ABB RobotStudio station: GJJRobotStudioAss1005f.rspag

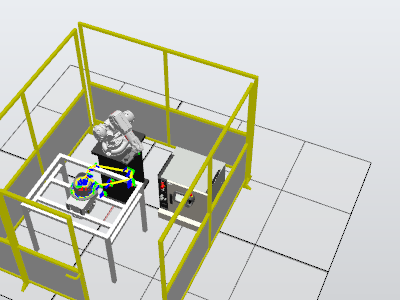
--- station ---
Station GJJAssessment1 (saved by RobotStudio 23.3.10550.0)
Controller Controller1
  mechanical unit ROB_1: IRB140_6_81_C_03, 6 joints, base frame (0, 0, 1000) mm
  mechanical unit M7DM1: MTD_250_M2009_REV1_01, 1 joints, base frame (769.44, 0, 1044.6) mm, rotated rx 0 ry 0 rz 180 deg
Layout (positions relative to the parent item):
  - IRB140_6_81_C_03 [mechanism, from %ABB.RobotStudio.Models.IRB140%\IRB140_6_81_C_G_03.rslib] at (0, 0, 1000) mm; joint values [-1.8898, -0.7873, -3.0781, -1.6729, -1.4587, 5.439] (rad or m)
  - MTD_250_M2009_REV1_01 [mechanism, from %ABB.RobotStudio.Models.GearUnits%\MTD_250_M2009_REV1_01.rslib] at (769.44, 0, 1044.6) mm, rotated rx 0 ry 0 rz 180 deg; joint values [19.7219] (rad or m)
  - potty1 [part] at (720.18, 192.49, 1031.85) mm, rotated rx 90 ry 0 rz 49.98 deg, size 275.1 x 194.8 x 257.3 mm
  - holder [part] at (392.98, 450, 1000) mm, rotated rx 90 ry 0 rz 0 deg, size 50 x 120 x 49.5 mm
  - SmartComponent_1_3 [smart component, from Libraries\SmartComponent_1.rslib] at (211.42, 435.22, 1354.55) mm, rotated rx -59.69 ry 89.8 rz -69.29 deg
      connections:
        SmartComponent_1_3.Closegrippers -> Attacher.Execute
        SmartComponent_1_3.Opengrippers -> Detacher.Execute
    - MyNewToolwithoutpen [mechanism, from Libraries\SmartComponent_1.rslib] at (0, 0, 0) mm
    - Attacher [smart component, from Components\Attacher.rslib]
        properties: Parent=MyNewToolwithoutpen; Flange=0; Child=The_Pen; Mount=false; Offset=[0 0 0]; Orientation=[0 0 0]
    - Detacher [smart component, from Components\Detacher.rslib]
        properties: Child=The_Pen; KeepPosition=false
  - The_Pen [part] at (215.35, 450.26, 1184.42) mm, rotated rx -90 ry 0 rz -90 deg, size 50 x 143 x 50 mm
  - Fence_2500 [graphiccomponentgroup, from Equipment\Fence_2500.rslib] at (1625.03, -938.91, 0) mm, rotated rx 0 ry 0 rz 90 deg
    - Body 1 [part, from Equipment\Fence_2500.rslib]
    - Body 2 [part, from Equipment\Fence_2500.rslib]
  - Fence_2500_2 [graphiccomponentgroup, from Equipment\Fence_2500.rslib] at (1620.42, 1504.32, 0) mm, rotated rx 0 ry 0 rz 90 deg
    - Body 1 [part, from Equipment\Fence_2500.rslib]
    - Body 2 [part, from Equipment\Fence_2500.rslib]
  - Fence_2500_3 [graphiccomponentgroup, from Equipment\Fence_2500.rslib] at (-975.12, -948, 0) mm
    - Body 1 [part, from Equipment\Fence_2500.rslib]
    - Body 2 [part, from Equipment\Fence_2500.rslib]
  - Gate [graphiccomponentgroup, from Equipment\Fence_Gate.rslib] at (1749.55, -943.09, 0) mm
    - Body 1 [part, from Equipment\Fence_Gate.rslib]
    - Body 2 [part, from Equipment\Fence_Gate.rslib]
    - Body 3 [part, from Equipment\Fence_Gate.rslib]
  - FlexPendant [part, from %ABB.RobotStudio.Models.IRC5%\FlexPendant.rslib] at (227.42, 1060.08, 778.08) mm, rotated rx -20.58 ry 0 rz 90 deg
  - MTDTable_Group [graphiccomponentgroup] at (367.09, -596.22, 0) mm
    - Height1 [part] at (850, 0, 0) mm, size 50 x 50 x 1000 mm
    - Height1_2 [part] at (850, 1150, 0) mm, size 50 x 50 x 1000 mm
    - Height1_3 [part] at (0, 1150, 0) mm, size 50 x 50 x 1000 mm
    - Height1_4 [part], size 50 x 50 x 1000 mm
    - Length1 [part] at (603.96, 0, 790) mm, size 50 x 1200 x 50 mm
    - Length1_2 [part] at (284.07, 0, 790) mm, size 50 x 1200 x 50 mm
    - Length1_3 [part] at (850, 0, 950) mm, size 50 x 1200 x 50 mm
    - Length1_4 [part] at (0, 0, 950) mm, size 50 x 1200 x 50 mm
    - Width1 [part] at (0, 0, 950) mm, size 900 x 50 x 50 mm
    - Width1_2 [part] at (0, 1150, 950) mm, size 900 x 50 x 50 mm
    - Width1_3 [part] at (0, 1150, 790) mm, size 900 x 50 x 50 mm
    - Width1_4 [part] at (0, 0, 790) mm, size 900 x 50 x 50 mm
  - IRC5_Singel-Cabinet [part, from %ABB.RobotStudio.Models.IRC5%\IRC5_Singel-Cabinet.rslib] at (-8.18, 1022.3, 100) mm, rotated rx 90 ry 0 rz 90 deg
  - RobotTable_Group [graphiccomponentgroup] at (-370.74, -2173.9, 0) mm
    - Bottom [part] at (0, 1929.69, 0) mm, size 550 x 500 x 50 mm
    - Top [part] at (0, 1929.69, 950) mm, size 550 x 500 x 50 mm
    - Table [part] at (46.03, 1981.79, 0) mm, size 450 x 400 x 1000 mm
Attachment: potty1 is attached to MTD_250_M2009_REV1_01 / Link1
Attachment: SmartComponent_1_3 is attached to IRB140_6_81_C_03 / Link6
Station logic (signal -> signal, property => property):
  Controller1.closegrips -> SmartComponent_1_3.Closegrippers
  Controller1.opengrips -> SmartComponent_1_3.Opengrippers

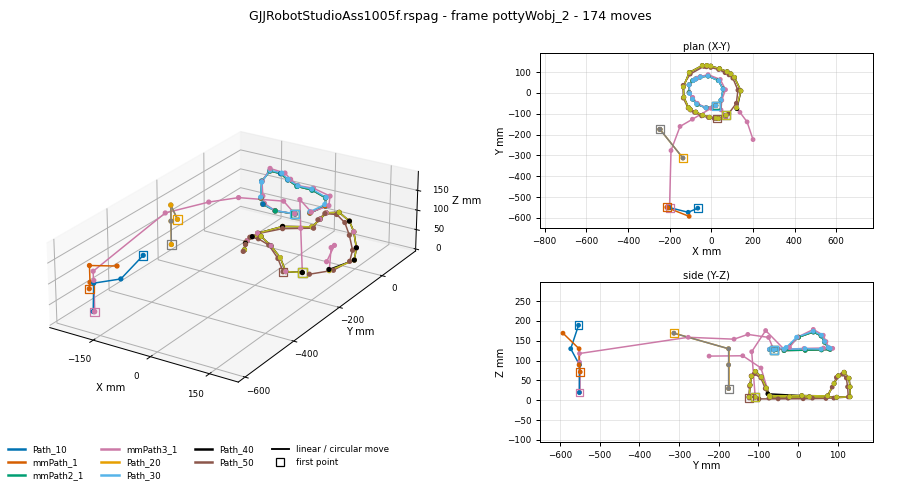
[picture p0: tool path of GJJRobotStudioAss1005f.rspag in frame pottyWobj_2, 174 of 175 moves have a stored position in this frame; points joined in program order, loops and branches not executed]
--- Controller Data/Controller1/RAPID/TASK1/PROGMOD/CalibData.mod ---
MODULE CalibData
    PERS tooldata MyNewTool1:=[TRUE,[[121,0,178],[1,0,0,0]],[2,[0,50,88],[1,0,0,0],0,0,0]];
    TASK PERS wobjdata pottyWobj_1:=[FALSE,FALSE,"M7DM1",[[-12.718015992,-112.561582584,1000],[0.69938504,0,0,0.714745106]],[[0,0,0],[1,0,0,0]]];
    PERS wobjdata pottyWobj_2:=[FALSE,FALSE,"M7DM1",[[0,0,1000],[1,0,0,0]],[[0,0,0],[1,0,0,0]]];
    PERS tooldata SmartTool:=[TRUE,[[121,0,178],[1,0,0,0]],[2,[0,50,88],[1,0,0,0],0,0,0]];
ENDMODULE

--- Controller Data/Controller1/RAPID/TASK1/PROGMOD/Module1.mod ---
MODULE Module1
        CONST robtarget Target_10:=[[22.32296581,-60.483962962,126.755003509],[0.000000091,-0.707106759,-0.000000134,0.707106804],[0,-2,1,0],[-27,9E+09,9E+09,9E+09,9E+09,9E+09]];
    CONST robtarget Target_20:=[[-24.392,-71.58,127.886],[0,-0.707106781,0,0.707106781],[0,-2,1,0],[-27,9E+09,9E+09,9E+09,9E+09,9E+09]];
    CONST robtarget Target_30:=[[-67.682,-54.97,128.901],[0,-0.707106781,0,0.707106781],[0,-2,1,0],[-27,9E+09,9E+09,9E+09,9E+09,9E+09]];
    CONST robtarget Target_40:=[[-89.149,-29.578,130.798],[0,-0.707106781,0,0.707106781],[0,-2,1,0],[-27,9E+09,9E+09,9E+09,9E+09,9E+09]];
    CONST robtarget Target_50:=[[-105.955,1.368,159.138],[0,-0.707106781,0,0.707106781],[-1,-3,2,0],[-27,9E+09,9E+09,9E+09,9E+09,9E+09]];
    CONST robtarget Target_60:=[[-106.053,38.886,172.329],[0,-0.707106781,0,0.707106781],[-1,-3,2,0],[-27,9E+09,9E+09,9E+09,9E+09,9E+09]];
    CONST robtarget Target_70:=[[-88.489,58.618,162.419],[0,-0.707106781,0,0.707106781],[-1,-3,2,0],[-27,9E+09,9E+09,9E+09,9E+09,9E+09]];
    CONST robtarget Target_80:=[[-73.57,67.289,146.688],[0,-0.707106781,0,0.707106781],[-1,-3,2,0],[-27,9E+09,9E+09,9E+09,9E+09,9E+09]];
    CONST robtarget Target_90:=[[-53.228,76.282,131.254],[0.030843565,-0.706433772,0.030843565,0.706433772],[-1,-3,2,0],[-27,9E+09,9E+09,9E+09,9E+09,9E+09]];
    CONST robtarget Target_100:=[[-14.851111209,80.984222238,128.595333376],[0.034268076,-0.706275937,0.034268076,0.706275937],[-1,-3,2,0],[-27,9E+09,9E+09,9E+09,9E+09,9E+09]];
    CONST robtarget Target_110:=[[34.482,59.302,127.342],[0.030843565,-0.706433772,0.030843565,0.706433772],[-1,-3,2,0],[-27,9E+09,9E+09,9E+09,9E+09,9E+09]];
    CONST robtarget Target_120:=[[57.63,18.266,126.328],[0.030843565,-0.706433772,0.030843565,0.706433772],[0,-2,1,0],[-27,9E+09,9E+09,9E+09,9E+09,9E+09]];
    CONST robtarget Target_130:=[[47.255,-35.047,125.605],[0.030843565,-0.706433772,0.030843565,0.706433772],[0,-2,1,0],[-27,9E+09,9E+09,9E+09,9E+09,9E+09]];
    CONST robtarget pTarget_1:=[[22.32296581,-60.483962962,126.755003509],[0.000000091,-0.707106759,-0.000000134,0.707106804],[0,-2,1,0],[-28.738330362,9E+09,9E+09,9E+09,9E+09,9E+09]];
    CONST robtarget pTarget_2:=[[-24.392,-71.58,127.886],[0,-0.707106781,0,0.707106781],[0,-2,1,0],[-28.261006609,9E+09,9E+09,9E+09,9E+09,9E+09]];
    CONST robtarget pTarget_3:=[[-67.682,-54.97,128.901],[0,-0.707106781,0,0.707106781],[0,-2,1,0],[-29.860701197,9E+09,9E+09,9E+09,9E+09,9E+09]];
    CONST robtarget pTarget_4:=[[-89.149,-29.578,130.798],[0,-0.707106781,0,0.707106781],[0,-2,1,0],[-32.019667198,9E+09,9E+09,9E+09,9E+09,9E+09]];
    CONST robtarget pTarget_5:=[[-105.955,1.368,159.138],[0,-0.707106781,0,0.707106781],[0,-2,1,0],[-33.289584297,9E+09,9E+09,9E+09,9E+09,9E+09]];
    CONST robtarget pTarget_6:=[[-106.053,38.886,172.329],[0,-0.707106781,0,0.707106781],[0,-2,1,0],[-35.350974752,9E+09,9E+09,9E+09,9E+09,9E+09]];
    CONST robtarget pTarget_7:=[[-88.489,58.618,162.419],[0,-0.707106781,0,0.707106781],[0,-2,1,0],[-36.641710687,9E+09,9E+09,9E+09,9E+09,9E+09]];
    CONST robtarget pTarget_8:=[[-73.57,67.289,146.688],[0,-0.707106781,0,0.707106781],[0,-2,1,0],[-37.385652325,9E+09,9E+09,9E+09,9E+09,9E+09]];
    CONST robtarget pTarget_9:=[[-53.228,76.282,131.254],[0.030843565,-0.706433772,0.030843565,0.706433772],[0,-2,1,0],[-33.888712133,9E+09,9E+09,9E+09,9E+09,9E+09]];
    CONST robtarget pTarget_10:=[[-14.851111209,80.984222238,128.595333376],[0.034268076,-0.706275937,0.034268076,0.706275937],[0,-2,1,0],[-32.382364491,9E+09,9E+09,9E+09,9E+09,9E+09]];
    CONST robtarget pTarget_11:=[[34.482,59.302,127.342],[0.030843565,-0.706433772,0.030843565,0.706433772],[0,-2,1,0],[-29.119527613,9E+09,9E+09,9E+09,9E+09,9E+09]];
    CONST robtarget pTarget_12:=[[57.63,18.266,126.328],[0.030843565,-0.706433772,0.030843565,0.706433772],[0,-2,1,0],[-25.00117949,9E+09,9E+09,9E+09,9E+09,9E+09]];
    CONST robtarget pTarget_13:=[[47.255,-35.047,125.605],[0.030843565,-0.706433772,0.030843565,0.706433772],[0,-2,1,0],[-20.912381123,9E+09,9E+09,9E+09,9E+09,9E+09]];
    CONST robtarget pTarget_14:=[[22.32296581,-60.483962962,126.755003509],[0.420603287,-0.568412565,0.420603132,0.568412734],[-2,-2,-1,7],[1152.182097091,9E+09,9E+09,9E+09,9E+09,9E+09]];
    CONST robtarget pTarget_15:=[[-24.392,-71.58,127.886],[0.560985527,-0.430459335,0.560985527,0.430459335],[-2,-2,-1,7],[1183.800837927,9E+09,9E+09,9E+09,9E+09,9E+09]];
    CONST robtarget pTarget_16:=[[-67.682,-54.97,128.901],[0.650895224,-0.276288631,0.650895224,0.276288631],[-2,-2,-1,7],[1212.326318879,9E+09,9E+09,9E+09,9E+09,9E+09]];
    CONST robtarget pTarget_17:=[[-89.149,-29.578,130.798],[0.674379723,-0.212631111,0.674379723,0.212631111],[-2,-2,-1,7],[1224.558462092,9E+09,9E+09,9E+09,9E+09,9E+09]];
    CONST robtarget pTarget_18:=[[-105.955,1.368,159.138],[0.704927007,-0.055478959,0.704927007,0.055478959],[-2,-2,-1,7],[1249.474772944,9E+09,9E+09,9E+09,9E+09,9E+09]];
    CONST robtarget pTarget_19:=[[-106.053,38.886,172.329],[0.668582596,0.230211451,0.668582596,-0.230211451],[-2,-2,-1,7],[1290.670999048,9E+09,9E+09,9E+09,9E+09,9E+09]];
    CONST robtarget pTarget_20:=[[-88.489,58.618,162.419],[0.59966056,0.374709505,0.59966056,-0.374709505],[-2,-2,-1,7],[1313.674902976,9E+09,9E+09,9E+09,9E+09,9E+09]];
    CONST robtarget pTarget_21:=[[-73.57,67.289,146.688],[0.593029646,0.385117955,0.593029646,-0.385117955],[-2,-2,-1,7],[1316.53427483,9E+09,9E+09,9E+09,9E+09,9E+09]];
    CONST robtarget pTarget_22:=[[-53.228,76.282,131.254],[0.529591668,0.46854313,0.529591668,-0.46854313],[-2,-2,-1,7],[1331.940227629,9E+09,9E+09,9E+09,9E+09,9E+09]];
    CONST robtarget pTarget_23:=[[-14.851111209,80.984222238,128.595333376],[0.397679767,0.584680086,0.397679767,-0.584680086],[-2,-2,-1,7],[1358.742450888,9E+09,9E+09,9E+09,9E+09,9E+09]];
    CONST robtarget pTarget_24:=[[34.482,59.302,127.342],[0.200829174,0.677987937,0.200829174,-0.677987937],[-2,-2,-1,7],[1392.934551377,9E+09,9E+09,9E+09,9E+09,9E+09]];
    CONST robtarget pTarget_25:=[[57.63,18.266,126.328],[0.03700711,-0.706137716,0.03700711,0.706137716],[-2,-2,-1,7],[1429.318516515,9E+09,9E+09,9E+09,9E+09,9E+09]];
    CONST robtarget pTarget_26:=[[47.255,-35.047,125.605],[0.247634015,-0.662327256,0.247634015,0.662327256],[-2,-2,-1,7],[1462.59869553,9E+09,9E+09,9E+09,9E+09,9E+09]];
    CONST robtarget pTarget_27:=[[21.661851249,-61.061928953,127.311494101],[0.275135891,-0.748199414,0.430396229,0.423387487],[-2,-1,2,7],[1139.702173994,9E+09,9E+09,9E+09,9E+09,9E+09]];
    CONST robtarget pTarget_28:=[[-25.541964022,-71.803453943,128.603323164],[0.398718476,-0.558872477,0.658088274,0.309200508],[-2,-2,3,7],[1178.047480316,9E+09,9E+09,9E+09,9E+09,9E+09]];
    CONST robtarget pTarget_29:=[[-67.001544905,-49.907510935,129.609796487],[0.477648278,-0.314235617,0.804160958,0.162583065],[-2,-2,3,7],[1214.859914174,9E+09,9E+09,9E+09,9E+09,9E+09]];
    CONST robtarget pTarget_30:=[[-88.863113938,-21.358868065,133.25648507],[0.496755294,-0.083191982,0.859967881,0.08227099],[-2,-2,3,7],[1237.862475165,9E+09,9E+09,9E+09,9E+09,9E+09]];
    CONST robtarget pTarget_31:=[[-103.66820786,-1.037658351,159.27905514],[0.503428696,0.041812518,0.862969924,0.009704173],[-2,-2,3,7],[1252.858728015,9E+09,9E+09,9E+09,9E+09,9E+09]];
    CONST robtarget pTarget_32:=[[-105.807495868,38.716134684,178.778669083],[0.497126729,0.194647881,0.841770342,-0.07999943],[-2,-2,3,7],[1272.269886237,9E+09,9E+09,9E+09,9E+09,9E+09]];
    CONST robtarget pTarget_33:=[[-79.758424949,63.871478291,164.023743839],[0.454575124,0.220893556,0.813153027,-0.288703392],[-2,-2,3,7],[1299.878587466,9E+09,9E+09,9E+09,9E+09,9E+09]];
    CONST robtarget pTarget_34:=[[-68.133139298,70.64610012,148.183864604],[0.402843516,0.319245262,0.758664918,-0.400283783],[-2,-2,3,7],[1325.452157679,9E+09,9E+09,9E+09,9E+09,9E+09]];
    CONST robtarget pTarget_35:=[[-52.066445826,78.369443131,132.809909287],[0.359440021,0.437605524,0.71989125,-0.401323889],[-2,-2,3,7],[1332.23286127,9E+09,9E+09,9E+09,9E+09,9E+09]];
    CONST robtarget pTarget_36:=[[-14.789886007,87.630950106,130.994726027],[0.265470303,0.572769809,0.613967324,-0.473818942],[-2,-2,3,7],[1356.644476016,9E+09,9E+09,9E+09,9E+09,9E+09]];
    CONST robtarget pTarget_37:=[[43.441222586,64.517531507,131.854066039],[0.062810486,0.753611532,0.359959298,-0.546400774],[-2,-2,3,7],[1399.421839859,9E+09,9E+09,9E+09,9E+09,9E+09]];
    CONST robtarget pTarget_38:=[[68.57410492,15.460031277,130.8018654],[0.039118795,-0.83507438,-0.151938344,0.527290469],[-2,-2,3,7],[1418.228466896,9E+09,9E+09,9E+09,9E+09,9E+09]];
    CONST robtarget pTarget_39:=[[50.607224577,-34.806962301,128.663583191],[0.141697123,-0.846613093,0.166564157,0.485205707],[-2,-2,3,7],[1444.123595497,9E+09,9E+09,9E+09,9E+09,9E+09]];
    CONST robtarget Target_140:=[[21.661851249,-61.061928953,127.311494101],[0.275135891,-0.748199414,0.430396229,0.423387487],[-2,0,1,7],[9E+09,9E+09,9E+09,9E+09,9E+09,9E+09]];
    CONST robtarget Target_150:=[[-25.541964022,-71.803453943,128.603323164],[0.398718476,-0.558872477,0.658088274,0.309200508],[-2,0,1,7],[9E+09,9E+09,9E+09,9E+09,9E+09,9E+09]];
    CONST robtarget Target_160:=[[-70.285360364,-53.207095098,129.609796487],[0.477648494,-0.314234551,0.804161375,0.162582432],[-2,0,1,7],[9E+09,9E+09,9E+09,9E+09,9E+09,9E+09]];
    CONST robtarget Target_170:=[[-89.593649912,-29.910618198,133.25648507],[0.496755079,-0.083194226,0.859967664,0.082272286],[-2,-1,2,7],[9E+09,9E+09,9E+09,9E+09,9E+09,9E+09]];
    CONST robtarget Target_180:=[[-103.374591435,-3.380233796,158.939956104],[0.503428757,0.04181791,0.862969663,0.009701029],[-2,-1,2,7],[9E+09,9E+09,9E+09,9E+09,9E+09,9E+09]];
    CONST robtarget Target_190:=[[-105.807279367,38.716726355,173.986835788],[0.497126505,0.194650235,0.841769798,-0.08000082],[-2,-1,2,7],[9E+09,9E+09,9E+09,9E+09,9E+09,9E+09]];
    CONST robtarget Target_200:=[[-85.751795988,59.344494411,164.023743839],[0.454573854,0.220897134,0.813152055,-0.288705392],[-2,-1,2,7],[9E+09,9E+09,9E+09,9E+09,9E+09,9E+09]];
    CONST robtarget Target_210:=[[-73.056396585,67.172311626,148.183864604],[0.402844024,0.3192443,0.758665323,-0.400283272],[-2,-1,2,7],[9E+09,9E+09,9E+09,9E+09,9E+09,9E+09]];
    CONST robtarget Target_220:=[[-51.497066964,76.593174921,132.809909287],[0.359439579,0.437606317,0.719890768,-0.401324285],[-2,-1,2,7],[9E+09,9E+09,9E+09,9E+09,9E+09,9E+09]];
    CONST robtarget Target_230:=[[-15.541181275,81.174606587,130.994726027],[0.265467859,0.572772976,0.613964369,-0.473820311],[-2,-1,2,7],[9E+09,9E+09,9E+09,9E+09,9E+09,9E+09]];
    CONST robtarget Target_240:=[[36.385958915,58.474764975,129.050592097],[0.062809522,0.753612166,0.35995797,-0.546400884],[-2,-1,2,7],[9E+09,9E+09,9E+09,9E+09,9E+09,9E+09]];
    CONST robtarget Target_250:=[[56.31796631,17.844450548,130.08172897],[0.039121263,-0.835075091,-0.151934435,0.527290286],[-2,-1,2,7],[9E+09,9E+09,9E+09,9E+09,9E+09,9E+09]];
    CONST robtarget Target_260:=[[46.938014575,-34.542826443,128.663583191],[0.141699063,-0.846612427,0.166567542,0.485205141],[-2,-1,2,7],[9E+09,9E+09,9E+09,9E+09,9E+09,9E+09]];
    CONST speeddata v450 :=[450,500,5000,1000];
    CONST speeddata v570 :=[570,500,5000,1000];
    CONST robtarget Target_270:=[[28.677076143,-123.104507167,5.867],[0.258041636,-0.658342247,0.258041636,0.658342247],[-2,-2,-1,7],[1486.28,9E+09,9E+09,9E+09,9E+09,9E+09]];
    CONST robtarget Target_280:=[[13.873762379,-121.964833712,35.53],[0.258041636,-0.658342247,0.258041636,0.658342247],[-2,-2,-1,7],[1486.28,9E+09,9E+09,9E+09,9E+09,9E+09]];
    CONST robtarget Target_290:=[[-13.234506345,-118.163908584,61.544],[0.258041636,-0.658342247,0.258041636,0.658342247],[-2,-2,-1,7],[1486.28,9E+09,9E+09,9E+09,9E+09,9E+09]];
    CONST robtarget Target_300:=[[-46.220645775,-110.309155024,66.748],[0.258041636,-0.658342247,0.258041636,0.658342247],[-2,-2,-1,7],[1486.28,9E+09,9E+09,9E+09,9E+09,9E+09]];
    CONST robtarget Target_310:=[[-79.84479739,-93.59531345,56.672],[0.258041636,-0.658342247,0.258041636,0.658342247],[-2,-2,-1,7],[1486.28,9E+09,9E+09,9E+09,9E+09,9E+09]];
    CONST robtarget Target_320:=[[-98.531465892,-82.520749156,29.589],[0.258041636,-0.658342247,0.258041636,0.658342247],[-2,-2,-1,7],[1486.28,9E+09,9E+09,9E+09,9E+09,9E+09]];
    CONST robtarget Target_330:=[[-110.776911108,-73.064012909,5.336],[0.258041636,-0.658342247,0.258041636,0.658342247],[-2,-2,-1,7],[1486.28,9E+09,9E+09,9E+09,9E+09,9E+09]];
    CONST robtarget Target_340:=[[-134.120369798,-24.865373702,5.301],[0.258041636,-0.658342247,0.258041636,0.658342247],[-2,-2,-1,7],[1486.28,9E+09,9E+09,9E+09,9E+09,9E+09]];
    CONST robtarget Target_350:=[[-134.50109961,36.384840411,5.417],[0.258041636,-0.658342247,0.258041636,0.658342247],[-2,-2,-1,7],[1486.28,9E+09,9E+09,9E+09,9E+09,9E+09]];
    CONST robtarget Target_360:=[[-100.79194611,90.447985177,5.651866703],[0.368441335,-0.603532089,0.368441335,0.603532089],[-2,-2,-1,7],[1486.28,9E+09,9E+09,9E+09,9E+09,9E+09]];
    CONST robtarget Target_370:=[[-35.67611117,126.944138099,8.438],[0.368441335,-0.603532089,0.368441335,0.603532089],[-2,-2,-1,7],[1486.28,9E+09,9E+09,9E+09,9E+09,9E+09]];
    CONST robtarget Target_380:=[[-22.888942806,125.161125136,34],[0.467646131,-0.530383914,0.467646131,0.530383914],[-2,-2,-1,7],[1486.28,9E+09,9E+09,9E+09,9E+09,9E+09]];
    CONST robtarget Target_390:=[[-2.295280651,122.030536685,56.144],[0.467646131,-0.530383914,0.467646131,0.530383914],[-2,-2,-1,7],[1486.28,9E+09,9E+09,9E+09,9E+09,9E+09]];
    CONST robtarget Target_400:=[[35.672255719,112.225347141,65.796],[0.467646131,-0.530383914,0.467646131,0.530383914],[-2,-2,-1,7],[1486.28,9E+09,9E+09,9E+09,9E+09,9E+09]];
    CONST robtarget Target_410:=[[66.653398852,96.93447646,57.659],[0.467646131,-0.530383914,0.467646131,0.530383914],[-2,-2,-1,7],[1486.28,9E+09,9E+09,9E+09,9E+09,9E+09]];
    CONST robtarget Target_420:=[[85.443607613,86.389644565,33.215],[0.467646131,-0.530383914,0.467646131,0.530383914],[-2,-2,-1,7],[1486.28,9E+09,9E+09,9E+09,9E+09,9E+09]];
    CONST robtarget Target_430:=[[103.725052621,70.653994676,4.664],[0.467646131,-0.530383914,0.467646131,0.530383914],[-2,-2,-1,7],[1486.28,9E+09,9E+09,9E+09,9E+09,9E+09]];
    CONST robtarget Target_440:=[[128.235268841,13.075190339,3.892],[0.467646131,-0.530383914,0.467646131,0.530383914],[-2,-2,-1,7],[1486.28,9E+09,9E+09,9E+09,9E+09,9E+09]];
    CONST robtarget Target_450:=[[120.62439913,-49.938185156,3.552],[0.467646131,-0.530383914,0.467646131,0.530383914],[-2,-2,-1,7],[1486.28,9E+09,9E+09,9E+09,9E+09,9E+09]];
    CONST robtarget Target_460:=[[84.597015616,-98.201424098,3.56],[0.467646131,-0.530383914,0.467646131,0.530383914],[-2,-2,-1,7],[1486.28,9E+09,9E+09,9E+09,9E+09,9E+09]];
    CONST robtarget Target_470:=[[71.242416009,-107.772557509,8.209025746],[0.174799862,-0.515700022,-0.259736463,0.797518317],[-2,-2,-1,7],[1441.688025702,9E+09,9E+09,9E+09,9E+09,9E+09]];
    CONST robtarget Target_480:=[[35.905948113,-123.287954848,8.208925718],[0.293919639,-0.549171075,-0.178383912,0.761709627],[-2,-2,-1,7],[1459.16292809,9E+09,9E+09,9E+09,9E+09,9E+09]];
    CONST robtarget Target_490:=[[19.451367662,-120.616645158,38.428092757],[0.362384291,-0.563189666,-0.127385422,0.731620106],[-2,-2,-1,7],[1469.66295058,9E+09,9E+09,9E+09,9E+09,9E+09]];
    CONST robtarget Target_500:=[[-7.986408069,-117.142699446,60.432915128],[0.454519479,-0.574978367,-0.053005187,0.678234746],[-2,-2,-1,7],[1484.618988485,9E+09,9E+09,9E+09,9E+09,9E+09]];
    CONST robtarget Target_510:=[[-40.852476478,-107.237602711,72.961104317],[0.555581701,-0.576155908,0.038131829,0.598263576],[-2,-2,-1,7],[1502.725983899,9E+09,9E+09,9E+09,9E+09,9E+09]];
    CONST robtarget Target_520:=[[-74.159519922,-92.21104678,58.834289491],[0.638742587,-0.563988854,0.123798781,0.508525655],[-2,-2,-1,7],[1519.913909059,9E+09,9E+09,9E+09,9E+09,9E+09]];
    CONST robtarget Target_530:=[[-100.465335377,-79.723532493,30.774048691],[0.68456961,-0.549515625,0.177318953,0.444921359],[-2,-2,-1,7],[1530.921004793,9E+09,9E+09,9E+09,9E+09,9E+09]];
    CONST robtarget Target_540:=[[-109.159858595,-70.189932793,8.660053159],[0.710591932,-0.538497415,0.208398656,0.402056763],[-2,-2,-1,7],[1537.713054187,9E+09,9E+09,9E+09,9E+09,9E+09]];
    CONST robtarget Target_550:=[[-131.528835523,-20.99432089,8.849858328],[0.775035672,-0.487450607,0.309517923,0.256729954],[-2,-2,-1,7],[1560.145034667,9E+09,9E+09,9E+09,9E+09,9E+09]];
    CONST robtarget Target_560:=[[-133.511408104,28.717103726,8.849882583],[0.807906658,-0.426083945,0.389694645,0.117802322],[-2,-2,-1,7],[1580.207977693,9E+09,9E+09,9E+09,9E+09,9E+09]];
    CONST robtarget Target_570:=[[-105.220016344,97.835804319,7.723567347],[0.811117358,-0.311995048,0.48586887,-0.093162022],[-2,-2,-1,7],[1609.904000959,9E+09,9E+09,9E+09,9E+09,9E+09]];
    CONST robtarget Target_580:=[[-42.772966601,131.265585239,8.849856155],[0.760323837,-0.17737289,0.54949825,-0.297486461],[-2,-2,-1,7],[1639.536967918,9E+09,9E+09,9E+09,9E+09,9E+09]];
    CONST robtarget Target_590:=[[-20.677226151,131.336434461,33.808612732],[0.731445583,-0.128717242,0.562886627,-0.362736648],[-2,-2,-1,7],[1649.555052261,9E+09,9E+09,9E+09,9E+09,9E+09]];
    CONST robtarget Target_600:=[[-2.302409671,128.688449933,55.6328306],[0.701351929,-0.085004597,0.571124856,-0.417966611],[-2,-2,-1,7],[1658.384977698,9E+09,9E+09,9E+09,9E+09,9E+09]];
    CONST robtarget Target_610:=[[39.965261731,116.533928321,70.693283731],[0.623269206,0.009854665,0.577332123,-0.527376529],[-2,-2,-1,7],[1677.271959913,9E+09,9E+09,9E+09,9E+09,9E+09]];
    CONST robtarget Target_620:=[[76.374170257,101.815008545,61.775734849],[0.533694448,0.09949785,0.568778849,-0.617868137],[-2,-2,-1,7],[1695.161044972,9E+09,9E+09,9E+09,9E+09,9E+09]];
    CONST robtarget Target_630:=[[94.583391815,91.17035861,42.256995319],[0.494072556,0.134819543,0.561455475,-0.6499875],[-2,-2,-1,7],[1702.321050316,9E+09,9E+09,9E+09,9E+09,9E+09]];
    CONST robtarget Target_640:=[[111.532176391,74.761142197,11.245391431],[0.429626525,0.187911969,0.545983247,-0.694271153],[-2,-2,-1,7],[1713.300060313,9E+09,9E+09,9E+09,9E+09,9E+09]];
    CONST robtarget Target_650:=[[142.420180078,9.734677329,11.779013759],[0.247276977,0.315428686,0.483645885,-0.778103784],[-2,-2,-1,7],[1741.539955408,9E+09,9E+09,9E+09,9E+09,9E+09]];
    CONST robtarget Target_660:=[[123.438259377,-75.949644716,16.328578229],[0.022726415,-0.457092552,-0.352810078,0.816134154],[-2,-2,-1,7],[1779.990027369,9E+09,9E+09,9E+09,9E+09,9E+09]];
    CONST robtarget pTarget_40:=[[71.242416009,-107.772557509,8.209025746],[0.174799862,-0.515700022,-0.259736463,0.797518317],[-2,-3,3,7],[1444.124,9E+09,9E+09,9E+09,9E+09,9E+09]];
    CONST robtarget pTarget_41:=[[35.905948113,-123.287954848,8.208925718],[0.293919639,-0.549171075,-0.178383912,0.761709627],[-2,-2,3,7],[1456.352650691,9E+09,9E+09,9E+09,9E+09,9E+09]];
    CONST robtarget pTarget_42:=[[19.451367662,-120.616645158,38.428092757],[0.362384291,-0.563189666,-0.127385422,0.731620106],[-2,-2,3,7],[1464.272899759,9E+09,9E+09,9E+09,9E+09,9E+09]];
    CONST robtarget pTarget_43:=[[-7.986408069,-117.142699446,60.432915128],[0.454519479,-0.574978367,-0.053005187,0.678234746],[-2,-2,3,7],[1476.221016405,9E+09,9E+09,9E+09,9E+09,9E+09]];
    CONST robtarget pTarget_44:=[[-40.852476478,-107.237602711,72.961104317],[0.555581701,-0.576155908,0.038131829,0.598263576],[-2,-2,3,7],[1490.985116549,9E+09,9E+09,9E+09,9E+09,9E+09]];
    CONST robtarget pTarget_45:=[[-74.159519922,-92.21104678,58.834289491],[0.638742587,-0.563988854,0.123798781,0.508525655],[-2,-2,3,7],[1505.487479049,9E+09,9E+09,9E+09,9E+09,9E+09]];
    CONST robtarget pTarget_46:=[[-100.465335377,-79.723532493,30.774048691],[0.68456961,-0.549515625,0.177318953,0.444921359],[-2,-2,3,7],[1515.408168731,9E+09,9E+09,9E+09,9E+09,9E+09]];
    CONST robtarget pTarget_47:=[[-109.159858595,-70.189932793,8.660053159],[0.710591932,-0.538497415,0.208398656,0.402056763],[-2,-2,3,7],[1520.063,9E+09,9E+09,9E+09,9E+09,9E+09]];
    CONST robtarget pTarget_48:=[[-131.528835523,-20.99432089,8.849858328],[0.775035672,-0.487450607,0.309517923,0.256729954],[-2,-2,3,7],[1539.369,9E+09,9E+09,9E+09,9E+09,9E+09]];
    CONST robtarget pTarget_49:=[[-133.511408104,28.717103726,8.849882583],[0.807906658,-0.426083945,0.389694645,0.117802322],[-2,-2,3,7],[1560.776,9E+09,9E+09,9E+09,9E+09,9E+09]];
    CONST robtarget pTarget_50:=[[-105.220016344,97.835804319,7.723567347],[0.811117358,-0.311995048,0.48586887,-0.093162022],[-2,-2,3,7],[1589.275,9E+09,9E+09,9E+09,9E+09,9E+09]];
    CONST robtarget pTarget_51:=[[-42.772966601,131.265585239,8.849856155],[0.760323837,-0.17737289,0.54949825,-0.297486461],[-2,-2,3,7],[1620.827,9E+09,9E+09,9E+09,9E+09,9E+09]];
    CONST robtarget pTarget_52:=[[-20.677226151,131.336434461,33.808612732],[0.731445583,-0.128717242,0.562886627,-0.362736648],[-2,-2,3,7],[1625.263,9E+09,9E+09,9E+09,9E+09,9E+09]];
    CONST robtarget pTarget_53:=[[-2.302409671,128.688449933,55.6328306],[0.701351929,-0.085004597,0.571124856,-0.417966611],[-2,-2,3,7],[1635.912,9E+09,9E+09,9E+09,9E+09,9E+09]];
    CONST robtarget pTarget_54:=[[39.965261731,116.533928321,70.693283731],[0.623269206,0.009854665,0.577332123,-0.527376529],[-2,-2,3,7],[1653.168,9E+09,9E+09,9E+09,9E+09,9E+09]];
    CONST robtarget pTarget_55:=[[76.374170257,101.815008545,61.775734849],[0.533694448,0.09949785,0.568778849,-0.617868137],[-2,-2,3,7],[1675.533,9E+09,9E+09,9E+09,9E+09,9E+09]];
    CONST robtarget pTarget_56:=[[94.583391815,91.17035861,42.256995319],[0.494072556,0.134819543,0.561455475,-0.6499875],[-2,-2,3,7],[1680.412,9E+09,9E+09,9E+09,9E+09,9E+09]];
    CONST robtarget pTarget_57:=[[111.532176391,74.761142197,11.245391431],[0.429626525,0.187911969,0.545983247,-0.694271153],[-2,-2,3,7],[1695.263,9E+09,9E+09,9E+09,9E+09,9E+09]];
    CONST robtarget pTarget_58:=[[142.420180078,9.734677329,11.779013759],[0.247276977,0.315428686,0.483645885,-0.778103784],[-2,-2,3,7],[1725.886,9E+09,9E+09,9E+09,9E+09,9E+09]];
    CONST robtarget pTarget_59:=[[121.905073811,-71.739532181,11.500213405],[0.022726415,-0.457092552,-0.352810078,0.816134154],[-2,-2,3,7],[1763.322,9E+09,9E+09,9E+09,9E+09,9E+09]];
    CONST robtarget Target_670:=[[-199.98149922,-551.012144001,19.625554326],[0.36593962,-0.605658715,0.367791709,0.60331996],[-2,-2,3,7],[1139.702085211,9E+09,9E+09,9E+09,9E+09,9E+09]];
    CONST robtarget Target_680:=[[-200.023621494,-550.89873014,118.000507691],[0.365939583,-0.605658706,0.367791685,0.603320006],[-2,-2,3,7],[1139.702085211,9E+09,9E+09,9E+09,9E+09,9E+09]];
    CONST robtarget pTarget_62:=[[-64.410782703,-553.340084227,189.267716418],[0.352589804,-0.613636494,0.350076493,0.613658808],[-2,-2,3,7],[1129.983608563,9E+09,9E+09,9E+09,9E+09,9E+09]];
    CONST robtarget pTarget_63:=[[-110.600377059,-573.078309502,130.015271631],[0.365938089,-0.605659551,0.367790209,0.603320964],[-2,-2,3,7],[1139.615002288,9E+09,9E+09,9E+09,9E+09,9E+09]];
    CONST robtarget pTarget_61:=[[70.602800442,-116.645993437,122.559935067],[0.174799851,-0.515700045,-0.259736445,0.79751831],[-2,-3,3,7],[1444.124,9E+09,9E+09,9E+09,9E+09,9E+09]];
    CONST robtarget pTarget_60:=[[47.00338421,-81.499598228,175.936341109],[0.073044799,-0.647210477,-0.244087052,0.718473776],[-2,-3,3,7],[1444.124,9E+09,9E+09,9E+09,9E+09,9E+09]];
    CONST robtarget Target_690:=[[-193.007269496,-276.732516219,158.890875708],[0.365939523,-0.605658674,0.367791751,0.603320035],[-2,-2,3,7],[1139.702085211,9E+09,9E+09,9E+09,9E+09,9E+09]];
    CONST robtarget Target_700:=[[-149.668443473,-161.170538978,154.148419387],[0.275135839,-0.748199499,0.430396198,0.423387403],[-2,-1,3,7],[1139.702173994,9E+09,9E+09,9E+09,9E+09,9E+09]];
    CONST robtarget Target_710:=[[-90.292046337,-126.476701138,166.180495482],[0.275135789,-0.748199443,0.430396221,0.423387512],[-2,-2,3,7],[1139.702173994,9E+09,9E+09,9E+09,9E+09,9E+09]];
    CONST robtarget Target_720:=[[-0.687749637,-74.120811069,158.609028152],[0.27513589,-0.748199434,0.430396304,0.423387376],[-2,-2,3,7],[1139.702173994,9E+09,9E+09,9E+09,9E+09,9E+09]];
    CONST robtarget Target_730:=[[137.93554063,-93.263146288,81.471338222],[0.022727287,-0.45709223,-0.352810038,0.816134328],[-2,-2,3,7],[1763.321961567,9E+09,9E+09,9E+09,9E+09,9E+09]];
    CONST robtarget Target_740:=[[172.14758438,-139.198510523,112.309481906],[0.26229043,0.60846551,0.186472977,-0.725397327],[-2,-2,3,7],[1763.321961567,9E+09,9E+09,9E+09,9E+09,9E+09]];
    CONST robtarget Target_750:=[[200.776272324,-224.144384668,111.45160635],[0.222338742,0.670021616,0.223996764,-0.671909196],[-2,-2,3,7],[1763.321961567,9E+09,9E+09,9E+09,9E+09,9E+09]];
    CONST robtarget Target_760:=[[-199.013784492,-550.767682807,95.923195322],[0.352589297,-0.613636341,0.350077136,0.613658885],[-2,-2,3,7],[1139.702,9E+09,9E+09,9E+09,9E+09,9E+09]];
    CONST robtarget Target_770:=[[-199.013734803,-550.767708125,20.299101051],[0.352589314,-0.613636402,0.350077056,0.61365886],[-2,-2,3,7],[1139.702,9E+09,9E+09,9E+09,9E+09,9E+09]];
    CONST robtarget Target_780:=[[-135.714251106,-312.89088919,169.267716418],[0.352589804,-0.613636494,0.350076493,0.613658808],[-2,-2,3,7],[1139.702,9E+09,9E+09,9E+09,9E+09,9E+09]];
    CONST robtarget Target_790:=[[-246.034064539,-174.869682836,130.015271631],[0.365939568,-0.605658649,0.367791694,0.603320067],[-2,-2,3,7],[1139.702,9E+09,9E+09,9E+09,9E+09,9E+09]];
    CONST robtarget Target_750_2:=[[392.813071448,453.37674407,1175.127145458],[0.707740314,-0.001805386,0.70647028,-0.000362333],[-2,-2,3,7],[1139.702,9E+09,9E+09,9E+09,9E+09,9E+09]];
    CONST robtarget Target_800:=[[-246.034087734,-174.869654102,89.321121536],[0.365939597,-0.60565863,0.36779173,0.603320046],[-2,-2,3,7],[1139.702,9E+09,9E+09,9E+09,9E+09,9E+09]];
    CONST robtarget Target_810:=[[-246.034068532,-174.869627009,29.625600669],[0.365939662,-0.605658616,0.367791752,0.603320008],[-2,-2,3,7],[1139.702,9E+09,9E+09,9E+09,9E+09,9E+09]];
    CONST robtarget pTarget_64:=[[-199.470008173,-550.949149016,89.321121536],[0.365939597,-0.60565863,0.36779173,0.603320046],[-2,-2,3,7],[1139.624399833,9E+09,9E+09,9E+09,9E+09,9E+09]];
    CONST robtarget pTarget_65:=[[-202.805135828,-551.347062425,19.625600669],[0.365939662,-0.605658616,0.367791752,0.603320008],[-2,-2,3,7],[1140.132499599,9E+09,9E+09,9E+09,9E+09,9E+09]];
    CONST robtarget Target_830:=[[-246.034049381,-174.869609723,130.015228039],[0.365939607,-0.605658611,0.367791711,0.603320071],[-2,-2,3,7],[1139.615002288,9E+09,9E+09,9E+09,9E+09,9E+09]];
    CONST robtarget Target_840:=[[-135.716232646,-312.890028555,169.267730844],[0.352591804,-0.613635407,0.350078464,0.613657622],[-2,-2,3,7],[1129.983982777,9E+09,9E+09,9E+09,9E+09,9E+09]];
    CONST robtarget Target_820:=[[-246.033087333,-174.871111423,89.321103246],[0.365937793,-0.605659752,0.367789909,0.603321125],[-2,-2,3,7],[1139.62405713,9E+09,9E+09,9E+09,9E+09,9E+09]];
    CONST robtarget pTarget_66:=[[-213.393171253,-549.002107498,71.430797059],[0.365939662,-0.605658616,0.367791752,0.603320008],[-2,-2,3,7],[1141.500072204,9E+09,9E+09,9E+09,9E+09,9E+09]];
    CONST robtarget pTarget_67:=[[-208.690497261,-551.97835733,89.321103246],[0.365937793,-0.605659752,0.367789909,0.603321125],[-2,-2,3,7],[1141.027520525,9E+09,9E+09,9E+09,9E+09,9E+09]];
    CONST robtarget pTarget_68:=[[-208.783243756,-551.985477169,130.015228039],[0.365939607,-0.605658611,0.367791711,0.603320071],[-2,-2,3,7],[1141.04074569,9E+09,9E+09,9E+09,9E+09,9E+09]];
    CONST robtarget pTarget_69:=[[-105.910603142,-592.632096271,169.267730844],[0.352591804,-0.613635407,0.350078464,0.613657622],[-2,-2,3,7],[1131.696892096,9E+09,9E+09,9E+09,9E+09,9E+09]];
!***********************************************************
    !
    ! Module:  Module1
    !
    ! Description:
    !   <Insert description here>
    !
    ! Author: sgjguo14
    !
    ! Version: 1.0
    !
    !***********************************************************


    !***********************************************************
    !
    ! Procedure main
    !
    !   This is the entry point of your program
    !
    !***********************************************************
    PROC main()
        ! Reset Clock
        ClkReset clock1;
        ! Start timing
        ClkStart clock1;

        ! Code to perform the task
        ActUnit M7DM1;
        mmPath3_2;
        WaitTime\InPos,0.5;
        CloseGripper;
        WaitTime\InPos,0.5;
        mmPath3_1;
        WaitTime\InPos,0.5;
        OpenGripper;
        mmPath3_3;
        DeactUnit M7DM1;

        ! Stop timing
        ClkStop clock1;
        ! Display the time on the FlexPendant
        TPWrite "Cycle Time="\Num:=ClkRead(clock1);
        ! Add a delay to display the time on the FlexPendant
        WaitTime\InPos, 1;
    ENDPROC

    PROC Path_10()
        ActUnit M7DM1;
        MoveL Target_10,v1000,z100,tool0\WObj:=pottyWobj_2;
        MoveL Target_20,v1000,z100,tool0\WObj:=pottyWobj_2;
        MoveL Target_30,v1000,z100,tool0\WObj:=pottyWobj_2;
        MoveL Target_40,v1000,z100,tool0\WObj:=pottyWobj_2;
        MoveL Target_50,v1000,z100,tool0\WObj:=pottyWobj_2;
        MoveL Target_60,v1000,z100,tool0\WObj:=pottyWobj_2;
        MoveL Target_70,v1000,z100,tool0\WObj:=pottyWobj_2;
        MoveL Target_80,v1000,z100,tool0\WObj:=pottyWobj_2;
        MoveL Target_90,v1000,z100,tool0\WObj:=pottyWobj_2;
        MoveL Target_100,v1000,z100,tool0\WObj:=pottyWobj_2;
        MoveL Target_110,v1000,z100,tool0\WObj:=pottyWobj_2;
        MoveL Target_120,v1000,z100,tool0\WObj:=pottyWobj_2;
        MoveL Target_130,v1000,z100,tool0\WObj:=pottyWobj_2;
        DeactUnit M7DM1;
    ENDPROC
    PROC mmPath_1()
        ActUnit M7DM1;
        MoveL pTarget_1,v1000,z100,tool0\WObj:=pottyWobj_2;
        MoveL pTarget_2,v1000,z100,tool0\WObj:=pottyWobj_2;
        MoveL pTarget_3,v1000,z100,tool0\WObj:=pottyWobj_2;
        MoveL pTarget_4,v1000,z100,tool0\WObj:=pottyWobj_2;
        MoveL pTarget_5,v1000,z100,tool0\WObj:=pottyWobj_2;
        MoveL pTarget_6,v1000,z100,tool0\WObj:=pottyWobj_2;
        MoveL pTarget_7,v1000,z100,tool0\WObj:=pottyWobj_2;
        MoveL pTarget_8,v1000,z100,tool0\WObj:=pottyWobj_2;
        MoveL pTarget_9,v1000,z100,tool0\WObj:=pottyWobj_2;
        MoveL pTarget_10,v1000,z100,tool0\WObj:=pottyWobj_2;
        MoveL pTarget_11,v1000,z100,tool0\WObj:=pottyWobj_2;
        MoveL pTarget_12,v1000,z100,tool0\WObj:=pottyWobj_2;
        MoveL pTarget_13,v1000,z100,tool0\WObj:=pottyWobj_2;
    ENDPROC
    PROC mmPath2_1()
        ActUnit M7DM1;
        MoveL pTarget_14,v1000,z100,tool0\WObj:=pottyWobj_2;
        MoveL pTarget_15,v1000,z100,tool0\WObj:=pottyWobj_2;
        MoveL pTarget_16,v1000,z100,tool0\WObj:=pottyWobj_2;
        MoveL pTarget_17,v1000,z100,tool0\WObj:=pottyWobj_2;
        MoveL pTarget_18,v1000,z100,tool0\WObj:=pottyWobj_2;
        MoveL pTarget_19,v1000,z100,tool0\WObj:=pottyWobj_2;
        MoveL pTarget_20,v1000,z100,tool0\WObj:=pottyWobj_2;
        MoveL pTarget_21,v1000,z100,tool0\WObj:=pottyWobj_2;
        MoveL pTarget_22,v1000,z100,tool0\WObj:=pottyWobj_2;
        MoveL pTarget_23,v1000,z100,tool0\WObj:=pottyWobj_2;
        MoveL pTarget_24,v1000,z100,tool0\WObj:=pottyWobj_2;
        MoveL pTarget_25,v1000,z100,tool0\WObj:=pottyWobj_2;
        MoveL pTarget_26,v1000,z100,tool0\WObj:=pottyWobj_2;
    ENDPROC
    PROC mmPath3_1()
        MoveL Target_670,v450,z100,SmartTool\WObj:=pottyWobj_2;
        MoveL Target_680,v450,z100,SmartTool\WObj:=pottyWobj_2;
        MoveL Target_690,v570,z100,SmartTool\WObj:=pottyWobj_2;
        MoveL Target_700,v570,z100,SmartTool\WObj:=pottyWobj_2;
        MoveL Target_710,v570,z100,SmartTool\WObj:=pottyWobj_2;
        MoveL Target_720,v450,z100,SmartTool\WObj:=pottyWobj_2;
        MoveL pTarget_27,v450,z100,SmartTool\WObj:=pottyWobj_2;
        MoveL pTarget_28,v450,z100,SmartTool\WObj:=pottyWobj_2;
        MoveL pTarget_29,v450,z100,SmartTool\WObj:=pottyWobj_2;
        MoveL pTarget_30,v450,z100,SmartTool\WObj:=pottyWobj_2;
        MoveL pTarget_31,v450,z100,SmartTool\WObj:=pottyWobj_2;
        MoveL pTarget_32,v450,z100,SmartTool\WObj:=pottyWobj_2;
        MoveL pTarget_33,v450,z100,SmartTool\WObj:=pottyWobj_2;
        MoveL pTarget_34,v450,z100,SmartTool\WObj:=pottyWobj_2;
        MoveL pTarget_35,v450,z100,SmartTool\WObj:=pottyWobj_2;
        MoveL pTarget_36,v450,z100,SmartTool\WObj:=pottyWobj_2;
        MoveL pTarget_37,v450,z100,SmartTool\WObj:=pottyWobj_2;
        MoveL pTarget_38,v450,z100,SmartTool\WObj:=pottyWobj_2;
        MoveL pTarget_39,v450,z100,SmartTool\WObj:=pottyWobj_2;
        MoveL pTarget_60,v450,z100,SmartTool\WObj:=pottyWobj_2;
        MoveL pTarget_61,v450,z100,SmartTool\WObj:=pottyWobj_2;
        MoveL pTarget_40,v450,z100,SmartTool\WObj:=pottyWobj_2;
        MoveL pTarget_41,v450,z100,SmartTool\WObj:=pottyWobj_2;
        MoveL pTarget_42,v450,z100,SmartTool\WObj:=pottyWobj_2;
        MoveL pTarget_43,v450,z100,SmartTool\WObj:=pottyWobj_2;
        MoveL pTarget_44,v450,z100,SmartTool\WObj:=pottyWobj_2;
        MoveL pTarget_45,v450,z100,SmartTool\WObj:=pottyWobj_2;
        MoveL pTarget_46,v450,z100,SmartTool\WObj:=pottyWobj_2;
        MoveL pTarget_47,v450,z100,SmartTool\WObj:=pottyWobj_2;
        MoveL pTarget_48,v450,z100,SmartTool\WObj:=pottyWobj_2;
        MoveL pTarget_49,v450,z100,SmartTool\WObj:=pottyWobj_2;
        MoveL pTarget_50,v450,z100,SmartTool\WObj:=pottyWobj_2;
        MoveL pTarget_51,v450,z100,SmartTool\WObj:=pottyWobj_2;
        MoveL pTarget_52,v450,z100,SmartTool\WObj:=pottyWobj_2;
        MoveL pTarget_53,v450,z100,SmartTool\WObj:=pottyWobj_2;
        MoveL pTarget_54,v450,z100,SmartTool\WObj:=pottyWobj_2;
        MoveL pTarget_55,v450,z100,SmartTool\WObj:=pottyWobj_2;
        MoveL pTarget_56,v450,z100,SmartTool\WObj:=pottyWobj_2;
        MoveL pTarget_57,v450,z100,SmartTool\WObj:=pottyWobj_2;
        MoveL pTarget_58,v450,z100,SmartTool\WObj:=pottyWobj_2;
        MoveL pTarget_59,v450,z100,SmartTool\WObj:=pottyWobj_2;
        MoveL Target_730,v450,z100,SmartTool\WObj:=pottyWobj_2;
        MoveL Target_740,v570,z100,SmartTool\WObj:=pottyWobj_2;
        MoveL Target_750,v570,z100,SmartTool\WObj:=pottyWobj_2;
        MoveL Target_750_2,v570,z100,SmartTool\WObj:=wobj0;
        MoveL Target_760,v450,z100,SmartTool\WObj:=pottyWobj_2;
        MoveL Target_770,v450,z100,SmartTool\WObj:=pottyWobj_2;
    ENDPROC
    PROC Path_20()
        MoveL Target_780,v450,z100,SmartTool\WObj:=pottyWobj_2;
        MoveL Target_790,v450,z100,SmartTool\WObj:=pottyWobj_2;
        MoveL Target_800,v450,z100,SmartTool\WObj:=pottyWobj_2;
        MoveL Target_810,v450,z100,SmartTool\WObj:=pottyWobj_2;

    ENDPROC
    PROC Path_30()
        MoveL Target_140,v1000,z100,tool0\WObj:=pottyWobj_2;
        MoveL Target_150,v1000,z100,tool0\WObj:=pottyWobj_2;
        MoveL Target_160,v1000,z100,tool0\WObj:=pottyWobj_2;
        MoveL Target_170,v1000,z100,tool0\WObj:=pottyWobj_2;
        MoveL Target_180,v1000,z100,tool0\WObj:=pottyWobj_2;
        MoveL Target_190,v1000,z100,tool0\WObj:=pottyWobj_2;
        MoveL Target_200,v1000,z100,tool0\WObj:=pottyWobj_2;
        MoveL Target_210,v1000,z100,tool0\WObj:=pottyWobj_2;
        MoveL Target_220,v1000,z100,tool0\WObj:=pottyWobj_2;
        MoveL Target_230,v1000,z100,tool0\WObj:=pottyWobj_2;
        MoveL Target_240,v1000,z100,tool0\WObj:=pottyWobj_2;
        MoveL Target_250,v1000,z100,tool0\WObj:=pottyWobj_2;
        MoveL Target_260,v1000,z100,tool0\WObj:=pottyWobj_2;

    ENDPROC
    PROC Path_40()
        MoveL Target_470,v1000,z100,tool0\WObj:=pottyWobj_2;
        MoveL Target_480,v1000,z100,tool0\WObj:=pottyWobj_2;
        MoveL Target_490,v1000,z100,tool0\WObj:=pottyWobj_2;
        MoveL Target_500,v1000,z100,tool0\WObj:=pottyWobj_2;
        MoveL Target_510,v1000,z100,tool0\WObj:=pottyWobj_2;
        MoveL Target_520,v1000,z100,tool0\WObj:=pottyWobj_2;
        MoveL Target_530,v1000,z100,tool0\WObj:=pottyWobj_2;
        MoveL Target_540,v1000,z100,tool0\WObj:=pottyWobj_2;
        MoveL Target_550,v1000,z100,tool0\WObj:=pottyWobj_2;
        MoveL Target_560,v1000,z100,tool0\WObj:=pottyWobj_2;
        MoveL Target_570,v1000,z100,tool0\WObj:=pottyWobj_2;
        MoveL Target_580,v1000,z100,tool0\WObj:=pottyWobj_2;
        MoveL Target_590,v1000,z100,tool0\WObj:=pottyWobj_2;
        MoveL Target_600,v1000,z100,tool0\WObj:=pottyWobj_2;
        MoveL Target_610,v1000,z100,tool0\WObj:=pottyWobj_2;
        MoveL Target_620,v1000,z100,tool0\WObj:=pottyWobj_2;
        MoveL Target_630,v1000,z100,tool0\WObj:=pottyWobj_2;
        MoveL Target_640,v1000,z100,tool0\WObj:=pottyWobj_2;
        MoveL Target_650,v1000,z100,tool0\WObj:=pottyWobj_2;
        MoveL Target_660,v1000,z100,tool0\WObj:=pottyWobj_2;
    ENDPROC
    PROC Path_50()
        MoveL Target_270,v1000,z100,tool0\WObj:=pottyWobj_2;
        MoveL Target_280,v1000,z100,tool0\WObj:=pottyWobj_2;
        MoveL Target_290,v1000,z100,tool0\WObj:=pottyWobj_2;
        MoveL Target_300,v1000,z100,tool0\WObj:=pottyWobj_2;
        MoveL Target_310,v1000,z100,tool0\WObj:=pottyWobj_2;
        MoveL Target_320,v1000,z100,tool0\WObj:=pottyWobj_2;
        MoveL Target_330,v1000,z100,tool0\WObj:=pottyWobj_2;
        MoveL Target_340,v1000,z100,tool0\WObj:=pottyWobj_2;
        MoveL Target_350,v1000,z100,tool0\WObj:=pottyWobj_2;
        MoveL Target_360,v1000,z100,tool0\WObj:=pottyWobj_2;
        MoveL Target_370,v1000,z100,tool0\WObj:=pottyWobj_2;
        MoveL Target_380,v1000,z100,tool0\WObj:=pottyWobj_2;
        MoveL Target_390,v1000,z100,tool0\WObj:=pottyWobj_2;
        MoveL Target_400,v1000,z100,tool0\WObj:=pottyWobj_2;
        MoveL Target_410,v1000,z100,tool0\WObj:=pottyWobj_2;
        MoveL Target_420,v1000,z100,tool0\WObj:=pottyWobj_2;
        MoveL Target_430,v1000,z100,tool0\WObj:=pottyWobj_2;
        MoveL Target_440,v1000,z100,tool0\WObj:=pottyWobj_2;
        MoveL Target_450,v1000,z100,tool0\WObj:=pottyWobj_2;
        MoveL Target_460,v1000,z100,tool0\WObj:=pottyWobj_2;
    ENDPROC
    PROC Path_60()
        MoveL Target_810,v450,z100,SmartTool\WObj:=pottyWobj_2;
        MoveL Target_820,v450,z100,SmartTool\WObj:=pottyWobj_2;
        MoveL Target_830,v450,z100,SmartTool\WObj:=pottyWobj_2;
        MoveL Target_840,v450,z100,SmartTool\WObj:=pottyWobj_2;
    ENDPROC
    PROC mmPath4_1()
        ActUnit M7DM1;
        MoveL pTarget_40,v1000,z100,tool0\WObj:=pottyWobj_2;
        MoveL pTarget_41,v1000,z100,tool0\WObj:=pottyWobj_2;
        MoveL pTarget_42,v1000,z100,tool0\WObj:=pottyWobj_2;
        MoveL pTarget_43,v1000,z100,tool0\WObj:=pottyWobj_2;
        MoveL pTarget_44,v1000,z100,tool0\WObj:=pottyWobj_2;
        MoveL pTarget_45,v1000,z100,tool0\WObj:=pottyWobj_2;
        MoveL pTarget_46,v1000,z100,tool0\WObj:=pottyWobj_2;
        MoveL pTarget_47,v1000,z100,tool0\WObj:=pottyWobj_2;
        MoveL pTarget_48,v1000,z100,tool0\WObj:=pottyWobj_2;
        MoveL pTarget_49,v1000,z100,tool0\WObj:=pottyWobj_2;
        MoveL pTarget_50,v1000,z100,tool0\WObj:=pottyWobj_2;
        MoveL pTarget_51,v1000,z100,tool0\WObj:=pottyWobj_2;
        MoveL pTarget_52,v1000,z100,tool0\WObj:=pottyWobj_2;
        MoveL pTarget_53,v1000,z100,tool0\WObj:=pottyWobj_2;
        MoveL pTarget_54,v1000,z100,tool0\WObj:=pottyWobj_2;
        MoveL pTarget_55,v1000,z100,tool0\WObj:=pottyWobj_2;
        MoveL pTarget_56,v1000,z100,tool0\WObj:=pottyWobj_2;
        MoveL pTarget_57,v1000,z100,tool0\WObj:=pottyWobj_2;
        MoveL pTarget_58,v1000,z100,tool0\WObj:=pottyWobj_2;
        MoveL pTarget_59,v1000,z100,tool0\WObj:=pottyWobj_2;
    ENDPROC
    PROC mmPath3_2()
        MoveL pTarget_62,v570,z100,SmartTool\WObj:=pottyWobj_2;
        MoveL pTarget_63,v570,z100,SmartTool\WObj:=pottyWobj_2;
        MoveL pTarget_64,v450,z100,SmartTool\WObj:=pottyWobj_2;
        MoveL pTarget_65,v450,z100,SmartTool\WObj:=pottyWobj_2;
    ENDPROC
    PROC mmPath3_3()
        MoveL pTarget_66,v450,z100,SmartTool\WObj:=pottyWobj_2;
        MoveL pTarget_67,v450,z100,SmartTool\WObj:=pottyWobj_2;
        MoveL pTarget_68,v570,z100,SmartTool\WObj:=pottyWobj_2;
        MoveL pTarget_69,v570,z100,SmartTool\WObj:=pottyWobj_2;
    ENDPROC
ENDMODULE

--- Controller Data/Controller1/RAPID/TASK1/SYSMOD/Grippers.sys ---
MODULE Grippers(SYSMODULE,READONLY)
    PROC OpenGripper()
        Reset closegrips;
        set opengrips;
    ENDPROC
    PROC CloseGripper()
        Reset opengrips;
        set closegrips;
    ENDPROC
ENDMODULE

--- Controller Data/Controller1/SYSPAR/EIO.cfg ---
EIO:CFG_1.0:6:1::
#
INDUSTRIAL_NETWORK:

      -Name "DeviceNet" -Label "DeviceNet Master/Slave Network" -Address "2"
#
DEVICENET_DEVICE:

      -Name "IOBoard" -Label "DeviceNet Generic Device" -VendorId 0\
      -ConnectionType "COS" -OutputSize -1 -InputSize -1
#
DEVICENET_INTERNAL_DEVICE:

      -Name "DN_Internal_Device" -VendorName "ABB Robotics"\
      -ProductName "DeviceNet Internal Slave Device"
#
EIO_SIGNAL:

      -Name "closegrips" -SignalType "DO" -Device "IOBoard"\
      -Label "Closes the gripper" -DeviceMap "0" -Access "All"

      -Name "opengrips" -SignalType "DO" -Device "IOBoard"\
      -Label "Opens the gripper" -DeviceMap "1" -Access "All"
